Yaskawa INFORM job: AIR_ONLY.JBI

/JOB
//NAME AIR_ONLY
//POS
///NPOS 0,0,0,0,0,0
//INST
///DATE 2022/12/12 13:29
///ATTR SC,RW
///GROUP1 RB1
///GROUP2 ST1
NOP
DOUT OT#(21) ON
TIMER T=0.10
DOUT OT#(21) OFF
DOUT OT#(17) ON
TIMER T=0.20
DOUT OT#(19) ON
TIMER T=5.00
DOUT OT#(19) OFF
TIMER T=0.30
DOUT OT#(17) OFF
DOUT OT#(23) ON
TIMER T=0.10
DOUT OT#(23) OFF
END
